FUNCTION_BLOCK "FB_Dual_Controller"   // FB2, SCL
{ S7_Optimized_Access := 'TRUE' }
VERSION : 1.0
// =============================================================================
//  TUSAÅž HGU Dual Controller V17
//  Purpose: Flow/Pressure control mode switching and coordination
//  Logic: IF Pressure â‰¤ 95% setpoint â†’ Flow control, ELSE Pressure limiting
//  Features: Seamless switching, motor RPM & valve current coordination
//  =============================================================================
   VAR_INPUT
      Enable : Bool := FALSE;   // Enable dual controller
      Motor_Enable : Bool := FALSE;   // Motor enable status Pressure inputs
      Pressure_Setpoint : Real := 280.0;   // Pressure setpoint (Bar)
      Pressure_Actual : Real := 0.0;   // Current pressure reading (Bar)
      Pressure_Threshold : Real := 95.0;   // Threshold percentage for mode switching Flow inputs
      Flow_Setpoint : Real := 30.0;   // Flow setpoint (L/min)
      Flow_Actual : Real := 0.0;   // Flow meter reading (L/min)
      Motor_Displacement : Real := 100.0;   // Motor displacement (cc/rev)
      Motor_Number : USInt := 1;   // Motor number (1-7) Control parameters
      Valve_Response_Time : Time := T#40MS;   // Valve response time Motor outputs
   END_VAR
   VAR_OUTPUT
      Motor_RPM : Real := 0.0;   // Motor RPM setpoint Valve outputs
      Valve_Current : Real := 0.0;   // Valve current setpoint (0-10000) Status outputs
      Flow_Control_Active : Bool := FALSE;   // Flow controller active
      Pressure_Control_Active : Bool := FALSE;   // Pressure controller active Error outputs
      Error_Status : Bool := FALSE;   // Error condition
      Error_Code : USInt := 0;   // Error code Controller instances
   END_VAR
   VAR
      Flow_Controller : "FB_Flow_Controller";   // Flow controller instance
      Pressure_Controller : "FB_Pressure_Controller";   // Pressure controller instance Control logic
      Control_Mode : USInt := 0;   // Control mode (0=Flow, 1=Pressure)
      Pressure_Limit : Real := 0.0;   // Calculated pressure limit
      Mode_Switch_Timer : TON_TIME;   // Mode switching delay timer
      Last_Mode : USInt := 0;   // Previous control mode Status tracking
      Last_Enable : Bool := FALSE;   // Previous enable state
      Startup_Timer : TON_TIME;   // Startup delay timer Error detection
      Controller_Error : Bool := FALSE;   // Controller error status
      Mode_Switch_Error : Bool := FALSE;   // Mode switching error
      Error_Timer : TON_TIME;   // Error persistence timer Mode change detection
      Mode_Change_Detected : Bool := FALSE;   // Mode change detection
   END_VAR
   VAR_TEMP
      Flow_Control_Enable : Bool;   // Flow controller enable
      Pressure_Control_Enable : Bool;   // Pressure controller enable
   END_VAR
   // Mode_Switch_Timer.PT := T#500MS;
   // Startup_Timer.PT := T#200MS;
   // Error_Timer.PT := T#1S;
BEGIN

   // =============================================================================
   // INITIALIZATION AND STARTUP
   // =============================================================================
   IF #Enable AND NOT #Last_Enable THEN
       // Reset all outputs on startup
       #Motor_RPM := 0.0;
       #Valve_Current := 0.0;
       #Control_Mode := 0;
       #Flow_Control_Active := FALSE;
       #Pressure_Control_Active := FALSE;
       #Error_Status := FALSE;
       #Error_Code := 0;
       #Last_Mode := 0;
       #Pressure_Limit := 0.0;
   END_IF;

   #Last_Enable := #Enable;

   // Startup delay (200ms for controller stabilization)
   #Startup_Timer(IN := #Enable,
                  PT := T#200ms);

   // =============================================================================
   // MAIN CONTROL LOGIC
   // =============================================================================
   IF #Enable AND #Motor_Enable AND #Startup_Timer.Q THEN

       // =============================================================================
       // CONTROL MODE DETERMINATION
       // =============================================================================
       #Pressure_Limit := #Pressure_Setpoint * (#Pressure_Threshold / 100.0);

       IF #Pressure_Actual <= #Pressure_Limit THEN
           // Pressure is below threshold - Use FLOW CONTROL
           #Control_Mode := 0;
           #Flow_Control_Enable := TRUE;
           #Pressure_Control_Enable := FALSE;
       ELSE
           // Pressure is above threshold - Use PRESSURE LIMITING
           #Control_Mode := 1;
           #Flow_Control_Enable := FALSE;
           #Pressure_Control_Enable := TRUE;
       END_IF;

       // =============================================================================
       // MODE SWITCHING DELAY (Prevent Oscillation)
       // =============================================================================
       IF #Control_Mode = #Last_Mode THEN
           #Mode_Change_Detected := 0;
       ELSE
           #Mode_Change_Detected := 1;
       END_IF;
       #Mode_Switch_Timer(IN := #Mode_Change_Detected,
                          PT := T#500ms);

       // Only apply mode change after delay
       IF NOT #Mode_Change_Detected OR #Mode_Switch_Timer.Q THEN
           #Last_Mode := #Control_Mode;

           // =============================================================================
           // FLOW CONTROLLER (Mode 0)
           // =============================================================================
           #Flow_Controller(
                            Enable := #Flow_Control_Enable,
                            Flow_Setpoint := #Flow_Setpoint,
                            Flow_Actual := #Flow_Actual,
                            Motor_Displacement := #Motor_Displacement,
                            Motor_Number := #Motor_Number,
                            Error_Threshold := 2.0,
                            Correction_Factor := 0.1,
                            Max_Correction := 50.0,
                            Max_RPM := 1500.0
           );

           // =============================================================================
           // PRESSURE CONTROLLER (Mode 1)
           // =============================================================================
           #Pressure_Controller(
                                Enable := #Pressure_Control_Enable,
                                Target_Pressure := #Pressure_Setpoint,
                                Current_Pressure := #Pressure_Actual,
                                Valve_Response_Time := #Valve_Response_Time,
                                Approach_Percentage := 10.0,
                                Tracking_Step_Size := 0.05,
                                Pressure_Threshold := #Pressure_Threshold
           );

           // =============================================================================
           // OUTPUT ASSIGNMENT BASED ON ACTIVE MODE
           // =============================================================================
           IF #Control_Mode = 0 THEN
               // FLOW CONTROL MODE
               #Motor_RPM := #Flow_Controller.Motor_RPM;
               #Valve_Current := 4000.0; // Base valve opening for flow control
               #Flow_Control_Active := #Flow_Controller.Control_Active;
               #Pressure_Control_Active := FALSE;
               #Controller_Error := #Flow_Controller.Error_Status;

           ELSE
               // PRESSURE LIMITING MODE
               #Motor_RPM := 0.0; // Reduce motor speed for pressure limiting
               #Valve_Current := #Pressure_Controller.Valve_Current;
               #Flow_Control_Active := FALSE;
               #Pressure_Control_Active := #Pressure_Controller.Control_Active;
               #Controller_Error := #Pressure_Controller.Error_Status;
           END_IF;

           // =============================================================================
           // ERROR HANDLING
           // =============================================================================
           IF #Controller_Error THEN
               #Error_Status := TRUE;
               IF #Control_Mode = 0 THEN
                   #Error_Code := #Flow_Controller.Error_Code + 10; // Flow controller errors: 11-14
               ELSE
                   #Error_Code := #Pressure_Controller.Error_Code + 20; // Pressure controller errors: 21-24
               END_IF;
           ELSE
               #Error_Status := FALSE;
               #Error_Code := 0;
           END_IF;
       ELSE 
           // Mode switching in progress - maintain previous outputs
           // This prevents output glitches during mode transitions
           ;
       END_IF;

   ELSE
       // =============================================================================
       // DISABLED STATE
       // =============================================================================
       #Motor_RPM := 0.0;
       #Valve_Current := 0.0;
       #Control_Mode := 0;
       #Flow_Control_Active := FALSE;
       #Pressure_Control_Active := FALSE;
       #Error_Status := FALSE;
       #Error_Code := 0;

       // Disable sub-controllers
       #Flow_Controller(
                        Enable := FALSE,
                        Flow_Setpoint := 0.0,
                        Flow_Actual := 0.0,
                        Motor_Displacement := #Motor_Displacement,
                        Motor_Number := #Motor_Number
       );
       #Pressure_Controller(
                            Enable := FALSE,
                            Target_Pressure := 0.0,
                            Current_Pressure := 0.0,
                            Valve_Response_Time := T#40ms
       );

       // Reset timers
       #Startup_Timer(IN := FALSE,
                      PT := T#200ms);
       #Mode_Switch_Timer(IN := FALSE,
                          PT := T#500ms);
       #Error_Timer(IN := FALSE,
                    PT := T#1s);
   END_IF;
END_FUNCTION_BLOCK

FUNCTION_BLOCK "FB_Flow_Controller"   // FB3, SCL
{ S7_Optimized_Access := 'TRUE' }
VERSION : 1.0
// =============================================================================
//  TUSAÅž HGU Flow Controller V17
//  Purpose: Flow-based motor RPM control with correction algorithm
//  Motor 1-6: Variable displacement (100cc), Motor 7: Fixed displacement
//  Features: Basic RPM calculation + fine-tuning correction
//  =============================================================================
   VAR_INPUT
      Enable : Bool := FALSE;   // Enable flow controller
      Flow_Setpoint : Real := 0.0;   // Target flow (L/min)
      Flow_Actual : Real := 0.0;   // Flow meter reading (L/min)
      Motor_Displacement : Real := 100.0;   // Motor displacement (cc/rev)
      Motor_Number : USInt := 1;   // Motor number (1-7) Correction algorithm parameters
      Error_Threshold : Real := 2.0;   // Â±2 L/min tolerance
      Correction_Factor : Real := 0.1;   // Correction gain (0.1 default)
      Max_Correction : Real := 50.0;   // Maximum RPM correction
      Max_RPM : Real := 1500.0;   // Maximum motor RPM
   END_VAR
   VAR_OUTPUT
      Motor_RPM : Real := 0.0;   // Calculated motor RPM
      Flow_Error : Real := 0.0;   // Flow error (L/min)
      Control_Active : Bool := FALSE;   // Controller active status
      Error_Status : Bool := FALSE;   // Error condition
      Error_Code : USInt := 0;   // Error code Internal calculations
   END_VAR
   VAR
      Basic_RPM : Real := 0.0;   // Basic RPM from flow setpoint
      Correction_RPM : Real := 0.0;   // RPM correction value
      Displacement_L_per_Rev : Real := 0.0;   // Displacement in L/rev Status tracking
      Last_Enable : Bool := FALSE;   // Previous enable state
      Startup_Timer : TON_TIME;   // Startup delay timer Error detection
      Flow_Error_Timer : TON_TIME;   // Flow error persistence timer
      Out_of_Range_Timer : TON_TIME;   // Out of range timer
   END_VAR
   VAR_TEMP
      Temp_RPM : Real;   // Temporary RPM calculation
      Temp_Error : Real;   // Temporary error calculation
   END_VAR
BEGIN

   // =============================================================================
   // INITIALIZATION AND STARTUP
   // =============================================================================
   IF #Enable AND NOT #Last_Enable THEN
       // Reset all outputs on startup
       #Motor_RPM := 0.0;
       #Flow_Error := 0.0;
       #Control_Active := FALSE;
       #Error_Status := FALSE;
       #Error_Code := 0;
       #Correction_RPM := 0.0;
   END_IF;

   #Last_Enable := #Enable;

   // Startup delay (100ms)
   #Startup_Timer(IN := #Enable,
                  PT := T#100ms);

   // =============================================================================
   // MAIN CONTROL LOGIC
   // =============================================================================
   IF #Enable AND #Startup_Timer.Q THEN

       // Convert displacement from cc/rev to L/rev
       #Displacement_L_per_Rev := #Motor_Displacement / 1000.0;

       // =============================================================================
       // BASIC RPM CALCULATION
       // =============================================================================
       IF #Displacement_L_per_Rev > 0.0 THEN
           #Basic_RPM := #Flow_Setpoint / #Displacement_L_per_Rev;
       ELSE
           #Basic_RPM := 0.0;
           #Error_Status := TRUE;
           #Error_Code := 1; // Invalid displacement
       END_IF;

       // =============================================================================
       // FLOW ERROR CALCULATION
       // =============================================================================
       #Flow_Error := #Flow_Setpoint - #Flow_Actual;

       // =============================================================================
       // CORRECTION ALGORITHM (Fine Tuning)
       // =============================================================================
       IF ABS(#Flow_Error) > #Error_Threshold THEN
           // Calculate correction based on error
           #Correction_RPM := #Flow_Error * #Correction_Factor;

           // Apply correction limits
           IF #Correction_RPM > #Max_Correction THEN
               #Correction_RPM := #Max_Correction;
           ELSIF #Correction_RPM < - #Max_Correction THEN
               #Correction_RPM := - #Max_Correction;
           END_IF;
       ELSE
           // Within tolerance - no correction needed
           #Correction_RPM := 0.0;
       END_IF;

       // =============================================================================
       // FINAL RPM CALCULATION
       // =============================================================================
       #Temp_RPM := #Basic_RPM + #Correction_RPM;

       // Apply motor limits
       IF #Temp_RPM > #Max_RPM THEN
           #Motor_RPM := #Max_RPM;
           #Error_Status := TRUE;
           #Error_Code := 2; // RPM limit exceeded
       ELSIF #Temp_RPM < 0.0 THEN
           #Motor_RPM := 0.0;
       ELSE
           #Motor_RPM := #Temp_RPM;
           #Error_Status := FALSE;
           #Error_Code := 0;
       END_IF;

       // =============================================================================
       // STATUS AND ERROR MONITORING
       // =============================================================================
       #Control_Active := TRUE;

       // Persistent flow error detection (>5 seconds)
       #Flow_Error_Timer(IN := (ABS(#Flow_Error) > (#Error_Threshold * 2.0)),
                         PT := T#5s);
       IF #Flow_Error_Timer.Q THEN
           #Error_Status := TRUE;
           #Error_Code := 3; // Persistent flow error
       END_IF;

       // Out of range detection
       #Out_of_Range_Timer(IN := (#Flow_Setpoint > (#Max_RPM * #Displacement_L_per_Rev)),
                           PT := T#1s);
       IF #Out_of_Range_Timer.Q THEN
           #Error_Status := TRUE;
           #Error_Code := 4; // Flow setpoint out of motor range
       END_IF;

   ELSE
       // =============================================================================
       // DISABLED STATE
       // =============================================================================
       #Motor_RPM := 0.0;
       #Flow_Error := 0.0;
       #Control_Active := FALSE;
       #Error_Status := FALSE;
       #Error_Code := 0;
       #Correction_RPM := 0.0;

       // Reset timers
       #Startup_Timer(IN := FALSE,
                      PT := T#100ms);
       #Flow_Error_Timer(IN := FALSE,
                         PT := T#2s);
       #Out_of_Range_Timer(IN := FALSE,
                           PT := T#1s);
   END_IF;
END_FUNCTION_BLOCK

FUNCTION_BLOCK "FB_Motor_Selection"   // FB4, SCL
{ S7_Optimized_Access := 'TRUE' }
VERSION : 1.0
// =============================================================================
//  TUSAÅž HGU Motor Selection V17
//  Purpose: Wear leveling algorithm for motor selection (Motors 1-6)
//  Features: Balanced wear, minimum motor count, maintenance tracking
//  Motor 7: Fixed displacement - separate control
//  =============================================================================
   VAR_INPUT
      Enable : Bool := FALSE;   // Enable motor selection
      Wear_Leveling_Enable : Bool := TRUE;   // Enable wear leveling algorithm
      Required_Total_Flow : Real := 0.0;   // Total required flow (L/min) Motor enable status (1-6)
      Motor_1_Enable : Bool := FALSE;
      Motor_2_Enable : Bool := FALSE;
      Motor_3_Enable : Bool := FALSE;
      Motor_4_Enable : Bool := FALSE;
      Motor_5_Enable : Bool := FALSE;
      Motor_6_Enable : Bool := FALSE;
      Motor_7_Enable : Bool := FALSE;   // Motor 7 separate Motor operating hours (1-6)
      Motor_1_Hours : Real := 0.0;
      Motor_2_Hours : Real := 0.0;
      Motor_3_Hours : Real := 0.0;
      Motor_4_Hours : Real := 0.0;
      Motor_5_Hours : Real := 0.0;
      Motor_6_Hours : Real := 0.0;   // Motor maintenance status (1-6)
      Motor_1_Maintenance_Due : Bool := FALSE;
      Motor_2_Maintenance_Due : Bool := FALSE;
      Motor_3_Maintenance_Due : Bool := FALSE;
      Motor_4_Maintenance_Due : Bool := FALSE;
      Motor_5_Maintenance_Due : Bool := FALSE;
      Motor_6_Maintenance_Due : Bool := FALSE;   // Safety status inputs (1-7)
      Pump_1_Line_Filter_Status : USInt := 2;
      Pump_1_Suction_Filter_Status : USInt := 1;
      Pump_1_Manual_Valve_Status : USInt := 1;
      Pump_2_Line_Filter_Status : USInt := 2;
      Pump_2_Suction_Filter_Status : USInt := 1;
      Pump_2_Manual_Valve_Status : USInt := 1;
      Pump_3_Line_Filter_Status : USInt := 2;
      Pump_3_Suction_Filter_Status : USInt := 1;
      Pump_3_Manual_Valve_Status : USInt := 1;
      Pump_4_Line_Filter_Status : USInt := 2;
      Pump_4_Suction_Filter_Status : USInt := 1;
      Pump_4_Manual_Valve_Status : USInt := 1;
      Pump_5_Line_Filter_Status : USInt := 2;
      Pump_5_Suction_Filter_Status : USInt := 1;
      Pump_5_Manual_Valve_Status : USInt := 1;
      Pump_6_Line_Filter_Status : USInt := 2;
      Pump_6_Suction_Filter_Status : USInt := 1;
      Pump_6_Manual_Valve_Status : USInt := 1;
      Pump_7_Line_Filter_Status : USInt := 2;
      Pump_7_Suction_Filter_Status : USInt := 1;
      Pump_7_Manual_Valve_Status : USInt := 1;   // System parameters
      Motor_Displacement : Real := 100.0;   // Motor displacement (cc/rev)
      Max_Motor_RPM : Real := 1500.0;   // Maximum motor RPM
      Motor_7_Fixed_Flow : Real := 34.0;   // Motor 7 fixed flow (L/min) Motor selection results (1-6)
   END_VAR
   VAR_OUTPUT
      Motor_1_Selected : Bool := FALSE;
      Motor_2_Selected : Bool := FALSE;
      Motor_3_Selected : Bool := FALSE;
      Motor_4_Selected : Bool := FALSE;
      Motor_5_Selected : Bool := FALSE;
      Motor_6_Selected : Bool := FALSE;
      Motor_7_Selected : Bool := FALSE;   // Motor 7 selection Selection information
      Selected_Motor_Count : USInt := 0;   // Number of selected motors
      Total_Available_Flow : Real := 0.0;   // Total available flow capacity
      Selection_Valid : Bool := FALSE;   // Selection is valid for required flow Error outputs
      Error_Status : Bool := FALSE;   // Error condition
      Error_Code : USInt := 0;   // Error code Initialize flag
   END_VAR
   VAR
      Init_Complete : Bool := FALSE;   // Initialization complete Motor selection arrays
      Motor_Available : Array[1..6] of Bool;   // Available motors (enabled & not in maintenance)
      Motor_Hours_Array : Array[1..6] of Real;   // Operating hours array
      Motor_Priority : Array[1..6] of USInt;   // Selection priority (0=highest)
      Motor_Selected_Array : Array[1..6] of Bool;   // Selected motors array Calculation variables
      Max_Flow_Per_Motor : Real := 0.0;   // Maximum flow per motor (L/min)
      Required_Motor_Count : USInt := 0;   // Required number of motors
      Available_Motor_Count : USInt := 0;   // Number of available motors
      Total_Required_Flow : Real := 0.0;   // Total flow including Motor 7 Wear leveling variables
      Min_Hours : Real := 0.0;   // Minimum operating hours
      Max_Hours : Real := 0.0;   // Maximum operating hours
      Temp_Hours : Real := 0.0;   // Temporary hours for sorting Loop counters
      i : USInt;
      j : USInt;
      k : USInt;
      Selected_Count : USInt;   // Status tracking
      Last_Enable : Bool := FALSE;   // Previous enable state
      Selection_Timer : TON_TIME;   // Selection calculation timer
   END_VAR
   VAR_TEMP
      Temp_Bool : Bool;   // Temporary boolean
      Temp_USInt : USInt;   // Temporary USInt
      Flow_Deficit : Real;   // Remaining flow to be covered
   END_VAR
BEGIN

   // Force initialization of outputs first
   #Motor_7_Selected := FALSE;

   // =============================================================================
   // INITIALIZATION
   // =============================================================================
   IF NOT #Init_Complete THEN
       // First-time initialization
       FOR #i := 1 TO 6 DO
           #Motor_Selected_Array[#i] := FALSE;
           #Motor_Available[#i] := FALSE;
           #Motor_Hours_Array[#i] := 0.0;
           #Motor_Priority[#i] := #i;
       END_FOR;
       #Motor_7_Selected := FALSE;
       #Selected_Motor_Count := 0;
       #Total_Available_Flow := 0.0;
       #Selection_Valid := FALSE;
       #Error_Status := FALSE;
       #Error_Code := 0;
       #Init_Complete := TRUE;
   END_IF;

   IF #Enable AND NOT #Last_Enable THEN
       // Reset all selections
       FOR #i := 1 TO 6 DO
           #Motor_Selected_Array[#i] := FALSE;
       END_FOR;
       #Motor_7_Selected := FALSE;
       #Selected_Motor_Count := 0;
       #Error_Status := FALSE;
       #Error_Code := 0;
   END_IF;

   #Last_Enable := #Enable;

   // =============================================================================
   // MAIN SELECTION ALGORITHM
   // =============================================================================
   IF #Enable THEN

       // =============================================================================
       // STEP 1: PREPARE MOTOR AVAILABILITY MATRIX WITH SAFETY CHECKS
       // =============================================================================

       // Motor 1 Safety Check
       #Motor_Available[1] := #Motor_1_Enable AND
       NOT #Motor_1_Maintenance_Due AND
       (#Pump_1_Line_Filter_Status <> 0) AND      // Line filter OK
       (#Pump_1_Suction_Filter_Status <> 0) AND   // Suction filter OK
       (#Pump_1_Manual_Valve_Status = 1);         // Manual valve open

       // Motor 2 Safety Check
       #Motor_Available[2] := #Motor_2_Enable AND
       NOT #Motor_2_Maintenance_Due AND
       (#Pump_2_Line_Filter_Status <> 0) AND      // Line filter OK
       (#Pump_2_Suction_Filter_Status <> 0) AND   // Suction filter OK
       (#Pump_2_Manual_Valve_Status = 1);         // Manual valve open

       // Motor 3 Safety Check
       #Motor_Available[3] := #Motor_3_Enable AND
       NOT #Motor_3_Maintenance_Due AND
       (#Pump_3_Line_Filter_Status <> 0) AND      // Line filter OK
       (#Pump_3_Suction_Filter_Status <> 0) AND   // Suction filter OK
       (#Pump_3_Manual_Valve_Status = 1);         // Manual valve open

       // Motor 4 Safety Check
       #Motor_Available[4] := #Motor_4_Enable AND
       NOT #Motor_4_Maintenance_Due AND
       (#Pump_4_Line_Filter_Status <> 0) AND      // Line filter OK
       (#Pump_4_Suction_Filter_Status <> 0) AND   // Suction filter OK
       (#Pump_4_Manual_Valve_Status = 1);         // Manual valve open

       // Motor 5 Safety Check
       #Motor_Available[5] := #Motor_5_Enable AND
       NOT #Motor_5_Maintenance_Due AND
       (#Pump_5_Line_Filter_Status <> 0) AND      // Line filter OK
       (#Pump_5_Suction_Filter_Status <> 0) AND   // Suction filter OK
       (#Pump_5_Manual_Valve_Status = 1);         // Manual valve open

       // Motor 6 Safety Check
       #Motor_Available[6] := #Motor_6_Enable AND
       NOT #Motor_6_Maintenance_Due AND
       (#Pump_6_Line_Filter_Status <> 0) AND      // Line filter OK
       (#Pump_6_Suction_Filter_Status <> 0) AND   // Suction filter OK
       (#Pump_6_Manual_Valve_Status = 1);         // Manual valve open

       #Motor_Hours_Array[1] := #Motor_1_Hours;
       #Motor_Hours_Array[2] := #Motor_2_Hours;
       #Motor_Hours_Array[3] := #Motor_3_Hours;
       #Motor_Hours_Array[4] := #Motor_4_Hours;
       #Motor_Hours_Array[5] := #Motor_5_Hours;
       #Motor_Hours_Array[6] := #Motor_6_Hours;

       // Count available motors
       #Available_Motor_Count := 0;
       FOR #i := 1 TO 6 DO
           IF #Motor_Available[#i] THEN
               #Available_Motor_Count := #Available_Motor_Count + 1;
           END_IF;
       END_FOR;

       // =============================================================================
       // STEP 2: CALCULATE FLOW REQUIREMENTS
       // =============================================================================
       #Max_Flow_Per_Motor := (#Max_Motor_RPM * #Motor_Displacement) / 1000.0; // L/min
       #Total_Required_Flow := #Required_Total_Flow;

       // Check if Motor 7 is needed and available
       IF #Motor_7_Enable AND (#Total_Required_Flow > 0.0) THEN
           #Motor_7_Selected := TRUE;
           #Total_Required_Flow := #Total_Required_Flow - #Motor_7_Fixed_Flow;
       ELSE
           #Motor_7_Selected := FALSE;
       END_IF;

       // Ensure non-negative flow requirement
       IF #Total_Required_Flow < 0.0 THEN
           #Total_Required_Flow := 0.0;
       END_IF;

       // Calculate required motor count for remaining flow
       IF #Total_Required_Flow > 0.0 THEN
           #Required_Motor_Count := REAL_TO_USINT(CEIL(#Total_Required_Flow / #Max_Flow_Per_Motor));
           IF #Required_Motor_Count > 6 THEN
               #Required_Motor_Count := 6; // Maximum 6 variable motors
           END_IF;
       ELSE
           #Required_Motor_Count := 0;
       END_IF;

       // =============================================================================
       // STEP 3: MOTOR SELECTION ALGORITHM
       // =============================================================================

       // Reset selection
       FOR #i := 1 TO 6 DO
           #Motor_Selected_Array[#i] := FALSE;
           #Motor_Priority[#i] := 99; // High number = low priority
       END_FOR;

       IF #Required_Motor_Count > 0 AND #Available_Motor_Count >= #Required_Motor_Count THEN

           IF #Wear_Leveling_Enable THEN
               // =============================================================================
               // WEAR LEVELING MODE: Select motors with least operating hours
               // =============================================================================

               // Assign priority based on operating hours (lower hours = higher priority)
               FOR #i := 1 TO 6 DO
                   IF #Motor_Available[#i] THEN
                       #Motor_Priority[#i] := 0; // Initialize as available
                   END_IF;
               END_FOR;

               // Sort available motors by operating hours (bubble sort)
               FOR #i := 1 TO 5 DO
                   FOR #j := #i + 1 TO 6 DO
                       IF #Motor_Available[#i] AND #Motor_Available[#j] THEN
                           IF #Motor_Hours_Array[#i] > #Motor_Hours_Array[#j] THEN
                               // Swap hours
                               #Temp_Hours := #Motor_Hours_Array[#i];
                               #Motor_Hours_Array[#i] := #Motor_Hours_Array[#j];
                               #Motor_Hours_Array[#j] := #Temp_Hours;

                               // Swap availability
                               #Temp_Bool := #Motor_Available[#i];
                               #Motor_Available[#i] := #Motor_Available[#j];
                               #Motor_Available[#j] := #Temp_Bool;
                           END_IF;
                       END_IF;
                   END_FOR;
               END_FOR;

               // Select required number of motors with lowest hours
               #Selected_Count := 0;
               FOR #i := 1 TO 6 DO
                   IF #Motor_Available[#i] AND #Selected_Count < #Required_Motor_Count THEN
                       #Motor_Selected_Array[#i] := TRUE;
                       #Selected_Count := #Selected_Count + 1;
                   END_IF;
               END_FOR;

           ELSE
               // =============================================================================
               // MANUAL MODE: Select first available motors
               // =============================================================================
               #Selected_Count := 0;
               FOR #i := 1 TO 6 DO
                   IF #Motor_Available[#i] AND #Selected_Count < #Required_Motor_Count THEN
                       #Motor_Selected_Array[#i] := TRUE;
                       #Selected_Count := #Selected_Count + 1;
                   END_IF;
               END_FOR;
           END_IF;

           #Selected_Motor_Count := #Selected_Count;

           // Check if selection is sufficient
           #Total_Available_Flow := USINT_TO_REAL(#Selected_Count) * #Max_Flow_Per_Motor;
           IF #Motor_7_Selected THEN
               #Total_Available_Flow := #Total_Available_Flow + #Motor_7_Fixed_Flow;
           END_IF;

           #Selection_Valid := (#Total_Available_Flow >= #Required_Total_Flow);

           IF NOT #Selection_Valid THEN
               #Error_Status := TRUE;
               #Error_Code := 1; // Insufficient motor capacity
           ELSE
               #Error_Status := FALSE;
               #Error_Code := 0;
           END_IF;

       ELSE
           // =============================================================================
           // ERROR CONDITIONS
           // =============================================================================
           #Selected_Motor_Count := 0;
           #Selection_Valid := FALSE;

           IF #Available_Motor_Count < #Required_Motor_Count THEN
               #Error_Status := TRUE;
               #Error_Code := 2; // Not enough available motors
           ELSE
               #Error_Status := FALSE;
               #Error_Code := 0;
           END_IF;
       END_IF;

       // =============================================================================
       // STEP 4: OUTPUT ASSIGNMENT
       // =============================================================================
       #Motor_1_Selected := #Motor_Selected_Array[1];
       #Motor_2_Selected := #Motor_Selected_Array[2];
       #Motor_3_Selected := #Motor_Selected_Array[3];
       #Motor_4_Selected := #Motor_Selected_Array[4];
       #Motor_5_Selected := #Motor_Selected_Array[5];
       #Motor_6_Selected := #Motor_Selected_Array[6];

   ELSE
       // =============================================================================
       // DISABLED STATE
       // =============================================================================
       #Motor_1_Selected := FALSE;
       #Motor_2_Selected := FALSE;
       #Motor_3_Selected := FALSE;
       #Motor_4_Selected := FALSE;
       #Motor_5_Selected := FALSE;
       #Motor_6_Selected := FALSE;
       #Motor_7_Selected := FALSE;

       #Selected_Motor_Count := 0;
       #Total_Available_Flow := 0.0;
       #Selection_Valid := FALSE;
       #Error_Status := FALSE;
       #Error_Code := 0;
   END_IF;
END_FUNCTION_BLOCK

FUNCTION_BLOCK "FB_Pressure_Controller"   // FB5, SCL
{ S7_Optimized_Access := 'TRUE' }
VERSION : 1.0
// =============================================================================
//  TUSAÅž HGU Pressure Controller V17
//  Purpose: Two-phase pressure control without PID
//  Phase 1: Lookup table fast approach (10% vicinity)
//  Phase 2: Time-based tracking for smooth transition
//  Features: Configurable response time, valve characteristic table
//  =============================================================================
   VAR_INPUT
      Enable : Bool := FALSE;   // Enable pressure controller
      Target_Pressure : Real := 280.0;   // Target pressure (Bar)
      Current_Pressure : Real := 0.0;   // Current pressure reading (Bar)
      Valve_Response_Time : Time := T#40MS;   // Valve response time (configurable) Algorithm parameters
      Approach_Percentage : Real := 10.0;   // Fast approach percentage (10%)
      Tracking_Step_Size : Real := 0.05;   // Tracking step size (5%)
      Pressure_Threshold : Real := 95.0;   // Pressure threshold for mode switching (95%)
   END_VAR
   VAR_OUTPUT
      Control_Phase : USInt := 0;   // Control phase (0=Disabled, 1=Approach, 2=Tracking)
      Control_Active : Bool := FALSE;   // Controller active status
      Error_Status : Bool := FALSE;   // Error condition
      Error_Code : USInt := 0;   // Error code Valve output (moved from VAR_OUTPUT for initialization)
   END_VAR
   VAR
      Valve_Current : Real := 0.0;   // Valve current setpoint (0-10000) Phase control
      Current_Phase : USInt := 0;   // Current control phase
      Approach_Target : Real := 0.0;   // Phase 1 approach target
      Last_Enable : Bool := FALSE;   // Previous enable state Timing control
      Phase_Timer : TON_TIME;   // Phase transition timer
      Tracking_Timer : TON_TIME;   // Tracking step timer
      Response_Timer : TON_TIME;   // Response delay timer Lookup table for pressure to current conversion Simple linear characteristic: 50-300 Bar -> 0-10000 Current
      Table_Min_Pressure : Real := 50.0;   // Minimum table pressure
      Table_Max_Pressure : Real := 300.0;   // Maximum table pressure
      Table_Min_Current : Real := 0.0;   // Minimum current output
      Table_Max_Current : Real := 10000.0;   // Maximum current output Error detection
      Pressure_Error : Real := 0.0;   // Pressure error
      Error_Timer : TON_TIME;   // Error persistence timer Step calculation
      Time_Step_Current : Real := 0.0;   // Time-based step current
      Previous_Current : Real := 0.0;   // Previous current value Internal initialization flag
      Init_Done : Bool := FALSE;   // Initialization complete flag
   END_VAR
   VAR_TEMP
      Temp_Current : Real;   // Temporary current calculation
      Pressure_Range : Real;   // Pressure range calculation
      Current_Range : Real;   // Current range calculation
      Normalized_Pressure : Real;   // Normalized pressure value
   END_VAR
   // Phase_Timer.PT := T#1S;
   // Tracking_Timer.PT := T#40MS;
   // Response_Timer.PT := T#40MS;
   // Error_Timer.PT := T#10S;
BEGIN

   // =============================================================================
   // INITIALIZATION AND STARTUP
   // =============================================================================
   IF NOT #Init_Done THEN
       // First-time initialization
       #Valve_Current := 0.0;
       #Control_Phase := 0;
       #Control_Active := FALSE;
       #Error_Status := FALSE;
       #Error_Code := 0;
       #Current_Phase := 1;
       #Previous_Current := 0.0;
       #Init_Done := TRUE;
   END_IF;

   IF #Enable AND NOT #Last_Enable THEN
       // Reset all outputs on startup
       #Valve_Current := 0.0;
       #Control_Phase := 0;
       #Control_Active := FALSE;
       #Error_Status := FALSE;
       #Error_Code := 0;
       #Current_Phase := 1; // Start with approach phase
       #Previous_Current := 0.0;
   END_IF;

   #Last_Enable := #Enable;

   // =============================================================================
   // MAIN CONTROL LOGIC
   // =============================================================================
   IF #Enable THEN

       // Calculate pressure error
       #Pressure_Error := #Target_Pressure - #Current_Pressure;

       // Check if pressure is above threshold (switch to pressure limiting)
       IF #Current_Pressure > (#Target_Pressure * #Pressure_Threshold / 100.0) THEN

           // =============================================================================
           // PHASE 1: FAST APPROACH (Lookup Table)
           // =============================================================================
           IF #Current_Phase = 1 THEN
               #Control_Phase := 1; // Approach phase

               // Calculate approach target (90% of the way to setpoint)
               IF #Current_Pressure < #Target_Pressure THEN
                   #Approach_Target := #Current_Pressure + (ABS(#Pressure_Error) * (100.0 - #Approach_Percentage) / 100.0);
               ELSE
                   #Approach_Target := #Current_Pressure - (ABS(#Pressure_Error) * (100.0 - #Approach_Percentage) / 100.0);
               END_IF;

               // Use lookup table to get current for approach target
               // Linear interpolation: 50-300 Bar -> 0-10000 Current
               IF #Approach_Target <= #Table_Min_Pressure THEN
                   #Valve_Current := #Table_Min_Current;
               ELSIF #Approach_Target >= #Table_Max_Pressure THEN
                   #Valve_Current := #Table_Max_Current;
               ELSE
                   #Normalized_Pressure := (#Approach_Target - #Table_Min_Pressure) / (#Table_Max_Pressure - #Table_Min_Pressure);
                   #Valve_Current := #Normalized_Pressure * #Table_Max_Current;
               END_IF;
               #Previous_Current := #Valve_Current;

               // Check if we're within 10% of target
               IF ABS(#Pressure_Error) <= (#Target_Pressure * #Approach_Percentage / 100.0) THEN
                   #Current_Phase := 2; // Switch to tracking phase
                   #Phase_Timer(IN := FALSE,
                                PT := T#1s); // Reset timer
               END_IF;

               // =============================================================================
               // PHASE 2: TIME-BASED TRACKING (Smooth Transition)
               // =============================================================================
           ELSIF #Current_Phase = 2 THEN
               #Control_Phase := 2; // Tracking phase

               // Time-based tracking with configurable response time
               #Tracking_Timer(IN := TRUE,
                               PT := #Valve_Response_Time);
               IF #Tracking_Timer.Q THEN
                   // Calculate step size based on remaining error
                   #Time_Step_Current := #Pressure_Error * #Tracking_Step_Size * 100.0; // Scale to current range

                   // Apply step to previous current
                   #Temp_Current := #Previous_Current + #Time_Step_Current;

                   // Limit current range
                   IF #Temp_Current > #Table_Max_Current THEN
                       #Valve_Current := #Table_Max_Current;
                   ELSIF #Temp_Current < #Table_Min_Current THEN
                       #Valve_Current := #Table_Min_Current;
                   ELSE
                       #Valve_Current := #Temp_Current;
                   END_IF;

                   #Previous_Current := #Valve_Current;
                   #Tracking_Timer(IN := FALSE,
                                   PT := #Valve_Response_Time); // Reset timer for next step
               END_IF;

           END_IF;

           #Control_Active := TRUE;

       ELSE
           // =============================================================================
           // PRESSURE BELOW THRESHOLD - FLOW CONTROL MODE
           // =============================================================================
           #Control_Phase := 0; // Flow control mode
           // Base opening calculation: 80% of target pressure
           #Temp_Current := #Target_Pressure * 0.8;
           IF #Temp_Current <= #Table_Min_Pressure THEN
               #Valve_Current := #Table_Min_Current;
           ELSIF #Temp_Current >= #Table_Max_Pressure THEN
               #Valve_Current := #Table_Max_Current;
           ELSE
               #Normalized_Pressure := (#Temp_Current - #Table_Min_Pressure) / (#Table_Max_Pressure - #Table_Min_Pressure);
               #Valve_Current := #Normalized_Pressure * #Table_Max_Current;
           END_IF;
           #Current_Phase := 1; // Reset to approach phase for next time
           #Control_Active := FALSE;
       END_IF;

       // =============================================================================
       // ERROR MONITORING
       // =============================================================================
       #Error_Timer(IN := (ABS(#Pressure_Error) > (#Target_Pressure * 0.2)),
                    PT := T#10s);
       IF #Error_Timer.Q THEN
           #Error_Status := TRUE;
           #Error_Code := 1; // Persistent pressure error
       ELSE
           #Error_Status := FALSE;
           #Error_Code := 0;
       END_IF;

   ELSE
       // =============================================================================
       // DISABLED STATE
       // =============================================================================
       #Valve_Current := 0.0;
       #Control_Phase := 0;
       #Control_Active := FALSE;
       #Error_Status := FALSE;
       #Error_Code := 0;
       #Current_Phase := 1; // Reset to approach phase

       // Reset all timers
       #Phase_Timer(IN := FALSE,
                    PT := T#1s);
       #Tracking_Timer(IN := FALSE,
                       PT := #Valve_Response_Time);
       #Response_Timer(IN := FALSE,
                       PT := #Valve_Response_Time);
       #Error_Timer(IN := FALSE,
                    PT := T#10s);
   END_IF;
END_FUNCTION_BLOCK

FUNCTION_BLOCK "FB_G120C_Drive"   // FB6, SCL
{ S7_Optimized_Access := 'TRUE' }
VERSION : 1.0
// =============================================================================
//  SIEMENS G120C Drive Controller for TUSAÅž HGU System
//  Purpose: 90kW G120C drive control with FREE telegram communication
//  Motors: 75kW hydraulic pump motors (6 units: Motor 1-6)
//  Communication: FREE telegram with RPM setpoint, status, diagnostics
//  
//  PROFINET Configuration:
//  Motor 1: IP 192.168.100.3, I/O Range: %QW100-%QW106 / %IW100-%IW106
//  Motor 2: IP 192.168.100.4, I/O Range: %QW110-%QW116 / %IW110-%IW116  
//  Motor 3: IP 192.168.100.5, I/O Range: %QW120-%QW126 / %IW120-%IW126
//  Motor 4: IP 192.168.100.6, I/O Range: %QW130-%QW136 / %IW130-%IW136
//  Motor 5: IP 192.168.100.7, I/O Range: %QW140-%QW146 / %IW140-%IW146
//  Motor 6: IP 192.168.100.8, I/O Range: %QW150-%QW156 / %IW150-%IW156
// 
//  FREE Telegram Structure (PZD-6/6 format):
//  SEND TO DRIVE (Control Data - %QW):
//    PZD[0] = Control Word       (%QW+0)  - Drive control bits
//    PZD[1] = Speed Setpoint     (%QW+2)  - RPM setpoint scaled
//    PZD[2] = Reserved           (%QW+4)  - Future use  
//    PZD[3] = Reserved           (%QW+6)  - Future use
//    PZD[4] = Reserved           (%QW+8)  - Future use
//    PZD[5] = Reserved           (%QW+10) - Future use
// 
//  RECEIVE FROM DRIVE (Status Data - %IW):
//    PZD[0] = Status Word        (%IW+0)  - Drive status bits
//    PZD[1] = Speed Actual       (%IW+2)  - RPM actual scaled  
//    PZD[2] = Current Actual     (%IW+4)  - Motor current scaled
//    PZD[3] = Temperature        (%IW+6)  - Motor temperature
//    PZD[4] = Error Word         (%IW+8)  - Error/warning codes
//    PZD[5] = Reserved           (%IW+10) - Future diagnostics
// 
//  Drive Parameter Setup (G120C commissioning):
//    P0918[0] = 6    ; FREE telegram, 6 PZD send
//    P0918[1] = 6    ; FREE telegram, 6 PZD receive  
//    P2079 = 3       ; PROFINET process data
//    P0922 = 1       ; Telegram 1 enable
//    P1000 = 1       ; Factory reset then set parameters
//  =============================================================================
   VAR_INPUT
      Enable : Bool := FALSE;   // Drive enable command
      Motor_Number : USInt := 1;   // Motor number (1-6) Control commands
      RPM_Setpoint : Real := 0.0;   // RPM setpoint (0-1500 RPM)
      Start_Command : Bool := FALSE;   // Start command (rising edge)
      Stop_Command : Bool := FALSE;   // Stop command (rising edge)
      Reset_Command : Bool := FALSE;   // Reset command (rising edge) Safety inputs
      Emergency_Stop : Bool := FALSE;   // Emergency stop input
      Motor_Enable_Switch : Bool := TRUE;   // Motor enable switch Configuration
      Max_RPM : Real := 1500.0;   // Maximum RPM limit
      Ramp_Up_Time : Time := T#5S;   // Acceleration time
      Ramp_Down_Time : Time := T#3S;   // Deceleration time Motor status
   END_VAR
   VAR_OUTPUT
      Motor_Running : Bool := FALSE;   // Motor running status
      Motor_Ready : Bool := FALSE;   // Motor ready status
      Motor_Fault : Bool := FALSE;   // Motor fault status Actual values
      RPM_Actual : Real := 0.0;   // Actual RPM
      Current_A : Real := 0.0;   // Motor current (Amperes)
      Temperature_C : Real := 0.0;   // Motor temperature (Celsius) Status and diagnostics
      Drive_Status : DWord := 0;   // Drive status word
      Error_Code : USInt := 0;   // Error code
      Warning_Code : USInt := 0;   // Warning code Command acknowledgments
      Start_Ack : Bool := FALSE;   // Start command acknowledged
      Stop_Ack : Bool := FALSE;   // Stop command acknowledged
      Reset_Ack : Bool := FALSE;   // Reset command acknowledged FREE telegram communication (to be mapped to G120C)
   END_VAR
   VAR_IN_OUT
      Control_Word : Word;   // Control word to drive
      Status_Word : Word;   // Status word from drive
      RPM_Setpoint_Word : Int;   // RPM setpoint to drive
      RPM_Actual_Word : Int;   // RPM actual from drive
      Current_Word : Int;   // Current from drive
      Temperature_Word : Int;   // Temperature from drive
      Error_Word : Word;   // Error word from drive Command processing
   END_VAR
   VAR
      Last_Start_Command : Bool := FALSE;   // Previous start command
      Last_Stop_Command : Bool := FALSE;   // Previous stop command
      Last_Reset_Command : Bool := FALSE;   // Previous reset command State machine
      Drive_State : USInt := 0;   // Drive state (0=Init, 1=Ready, 2=Running, 3=Fault)
      State_Timer : TON_TIME;   // State transition timer Command timers
      Start_Timer : TON_TIME;   // Start command timeout
      Stop_Timer : TON_TIME;   // Stop command timeout
      Reset_Cmd_Timer : TON_TIME;   // Reset command timeout Safety and monitoring
      Emergency_Stop_Delay : TON_TIME;   // Emergency stop delay timer
      Fault_Reset_Delay : TON_TIME;   // Fault reset delay timer
      Watchdog_Timer : TON_TIME;   // Communication watchdog timer Scaling and conversion
      RPM_Scale_Factor : Real := 10.0;   // RPM scaling (1500 RPM = 15000 in telegram)
      Current_Scale_Factor : Real := 0.1;   // Current scaling (100A = 1000 in telegram)
      Temperature_Offset : Real := 40.0;   // Temperature offset (Â°C) Internal flags
      Init_Complete : Bool := FALSE;   // Initialization complete
      Communication_OK : Bool := FALSE;   // Communication status
      Last_Enable : Bool := FALSE;   // Previous enable state Error tracking
      Communication_Error : Bool := FALSE;   // Communication error
      Parameter_Error : Bool := FALSE;   // Parameter error
      Safety_Error : Bool := FALSE;   // Safety error
   END_VAR
   VAR_TEMP
      Temp_RPM : Real;   // Temporary RPM calculation
      Temp_Status : Word;   // Temporary status processing
      Control_Bits : Word;   // Control word bits
   END_VAR
BEGIN

   // =============================================================================
   // INITIALIZATION
   // =============================================================================
   IF NOT #Init_Complete THEN
       // Initialize all outputs
       #Motor_Running := FALSE;
       #Motor_Ready := FALSE;
       #Motor_Fault := FALSE;
       #RPM_Actual := 0.0;
       #Current_A := 0.0;
       #Temperature_C := 0.0;
       #Drive_Status := 0;
       #Error_Code := 0;
       #Warning_Code := 0;

       // Initialize communication
       #Control_Word := 0;
       #RPM_Setpoint_Word := 0;

       // Initialize timers
       #Start_Timer(IN := FALSE,
                    PT := T#1s);
       #Stop_Timer(IN := FALSE,
                   PT := T#1s);
       #Reset_Cmd_Timer(IN := FALSE,
                        PT := T#1s);
       #Emergency_Stop_Delay(IN := FALSE,
                             PT := T#100ms);
       #State_Timer(IN := FALSE,
                    PT := T#2s);
       #Watchdog_Timer(IN := FALSE,
                       PT := T#5s);

       #Drive_State := 0;
       #Init_Complete := TRUE;
   END_IF;

   IF #Enable AND NOT #Last_Enable THEN
       // Reset on enable
       #Drive_State := 0;
       #Error_Code := 0;
       #Warning_Code := 0;
   END_IF;

   #Last_Enable := #Enable;

   // =============================================================================
   // MAIN CONTROL LOGIC
   // =============================================================================
   IF #Enable THEN

       // =============================================================================
       // SAFETY MONITORING
       // =============================================================================
       #Emergency_Stop_Delay(IN := #Emergency_Stop,
                             PT := T#100ms);
       #Safety_Error := #Emergency_Stop_Delay.Q OR NOT #Motor_Enable_Switch;

       // =============================================================================
       // COMMUNICATION PROCESSING
       // =============================================================================

       // Process status word from drive
       #Temp_Status := #Status_Word;
       #Motor_Ready := (#Temp_Status.%X0);         // Bit 0: Ready
       #Motor_Running := (#Temp_Status.%X2);       // Bit 2: Running  
       #Motor_Fault := (#Temp_Status.%X3);         // Bit 3: Fault
       #Communication_OK := (#Temp_Status.%X15);   // Bit 15: Communication OK

       // Process actual values from drive
       #RPM_Actual := INT_TO_REAL(#RPM_Actual_Word) / #RPM_Scale_Factor;
       #Current_A := INT_TO_REAL(#Current_Word) * #Current_Scale_Factor;
       #Temperature_C := INT_TO_REAL(#Temperature_Word) + #Temperature_Offset;

       // Drive status and error processing
       #Drive_Status := WORD_TO_DWORD(#Status_Word);
       IF #Error_Word > 0 THEN
           #Error_Code := WORD_TO_USINT(#Error_Word AND 16#00FF);
           #Warning_Code := WORD_TO_USINT((#Error_Word AND 16#FF00) / 256);
       ELSE
           #Error_Code := 0;
           #Warning_Code := 0;
       END_IF;

       // =============================================================================
       // COMMAND PROCESSING (RISING EDGE DETECTION)
       // =============================================================================

       // Timer calls - TIA Portal V17 compliant
       #Start_Timer(IN := (#Start_Command AND NOT #Last_Start_Command),
                    PT := T#1s);
       #Stop_Timer(IN := (#Stop_Command AND NOT #Last_Stop_Command),
                   PT := T#1s);
       #Reset_Cmd_Timer(IN := (#Reset_Command AND NOT #Last_Reset_Command),
                        PT := T#1s);

       // Command bit processing
       IF #Start_Command AND NOT #Last_Start_Command THEN
           #Control_Bits.%X0 := TRUE;              // Set start bit
       END_IF;

       IF #Stop_Command AND NOT #Last_Stop_Command THEN
           #Control_Bits.%X1 := TRUE;              // Set stop bit
       END_IF;

       IF #Reset_Command AND NOT #Last_Reset_Command THEN
           #Control_Bits.%X7 := TRUE;              // Set reset bit
       END_IF;

       // Update last command states
       #Last_Start_Command := #Start_Command;
       #Last_Stop_Command := #Stop_Command;
       #Last_Reset_Command := #Reset_Command;

       // =============================================================================
       // RPM SETPOINT PROCESSING
       // =============================================================================

       // Limit and scale RPM setpoint
       IF #RPM_Setpoint > #Max_RPM THEN
           #Temp_RPM := #Max_RPM;
       ELSIF #RPM_Setpoint < 0.0 THEN
           #Temp_RPM := 0.0;
       ELSE
           #Temp_RPM := #RPM_Setpoint;
       END_IF;

       // Convert to telegram format
       #RPM_Setpoint_Word := REAL_TO_INT(#Temp_RPM * #RPM_Scale_Factor);

       // =============================================================================
       // DRIVE STATE MACHINE
       // =============================================================================
       #State_Timer(IN := TRUE,
                    PT := T#2s);

       CASE #Drive_State OF
           0: // Initialization
               IF #State_Timer.Q THEN
                   IF #Communication_OK AND NOT #Safety_Error THEN
                       #Drive_State := 1;
                   END_IF;
                   #State_Timer(IN := FALSE,
                                PT := T#2s);
               END_IF;

           1: // Ready
               IF #Motor_Fault OR #Safety_Error THEN
                   #Drive_State := 3;
               ELSIF #Motor_Running THEN
                   #Drive_State := 2;
               END_IF;

           2: // Running
               IF #Motor_Fault OR #Safety_Error THEN
                   #Drive_State := 3;
               ELSIF NOT #Motor_Running THEN
                   #Drive_State := 1;
               END_IF;

           3: // Fault
               IF NOT #Motor_Fault AND NOT #Safety_Error AND #Reset_Cmd_Timer.Q THEN
                   #Drive_State := 1;
               END_IF;
       END_CASE;

       // =============================================================================
       // CONTROL WORD GENERATION
       // =============================================================================

       // Emergency stop override
       IF #Safety_Error THEN
           #Control_Word := 0;                     // Emergency stop - all bits off
       ELSE
           // Enable bit
           #Control_Bits.%X15 := TRUE;             // Drive enable

           // Copy control bits to control word
           #Control_Word := #Control_Bits;
       END_IF;

       // =============================================================================
       // COMMAND ACKNOWLEDGMENTS
       // =============================================================================
       // Timer outputs already called in command processing section
       #Start_Ack := #Start_Timer.Q AND #Motor_Running;
       #Stop_Ack := #Stop_Timer.Q AND NOT #Motor_Running;
       #Reset_Ack := #Reset_Cmd_Timer.Q AND NOT #Motor_Fault;

       // =============================================================================
       // ERROR MONITORING
       // =============================================================================

       // Communication watchdog
       #Watchdog_Timer(IN := NOT #Communication_OK,
                       PT := T#5s);
       #Communication_Error := #Watchdog_Timer.Q;

       // Parameter validation
       #Parameter_Error := (#Max_RPM <= 0.0) OR (#RPM_Scale_Factor <= 0.0);

   ELSE
       // =============================================================================
       // DISABLED STATE
       // =============================================================================
       #Motor_Running := FALSE;
       #Motor_Ready := FALSE;
       #RPM_Actual := 0.0;
       #Current_A := 0.0;
       #Drive_State := 0;

       // Reset all commands and timers
       #Control_Word := 0;
       #RPM_Setpoint_Word := 0;

       #Start_Timer(IN := FALSE,
                    PT := T#1s);
       #Stop_Timer(IN := FALSE,
                   PT := T#1s);
       #Reset_Cmd_Timer(IN := FALSE,
                        PT := T#1s);
       #State_Timer(IN := FALSE,
                    PT := T#2s);
       #Emergency_Stop_Delay(IN := FALSE,
                             PT := T#100ms);
       #Fault_Reset_Delay(IN := FALSE,
                          PT := T#500ms);
       #Watchdog_Timer(IN := FALSE,
                       PT := T#5s);

       #Start_Ack := FALSE;
       #Stop_Ack := FALSE;
       #Reset_Ack := FALSE;
   END_IF;
END_FUNCTION_BLOCK

ORGANIZATION_BLOCK "OB1"   // OB1, SCL, ProgramCycle
TITLE = 'Main Program OB1'
{ S7_Optimized_Access := 'FALSE' }
AUTHOR : TUSAS
FAMILY : Main
NAME : Main
VERSION : 3.0
// =============================================================================
//  MAIN ORGANIZATION BLOCK - V17 ARCHITECTURE
//  TIA Portal S7-1500 Structured Control Language (SCL)
//  Description: Simple system coordination calling FB_System_Coordinator
//  =============================================================================
   VAR_TEMP
      SystemStatus : DInt;   // 4 bytes
      CycleTime : Time;   // 4 bytes
      Reserved1 : DInt;   // 4 bytes
      Reserved2 : DInt;   // 4 bytes
      Reserved3 : DInt;   // 4 bytes
   END_VAR
BEGIN

   // =============================================================================
   // MAIN SYSTEM COORDINATION
   // =============================================================================

   // Call main system coordinator with minimal configuration
   "DB_System_Coordinator_Instance"(
                                    Enable := TRUE,
                                    SystemCommand := 1,
                                    System_Total_Flow_Setpoint := 100.0
   );
END_ORGANIZATION_BLOCK